FUNCTION_BLOCK Stage21 (* Template for a Basic Function Block Type *)
  (* Standard: 61499-2 *)
  (* Version 1.0, 2021-06-20, HP *)
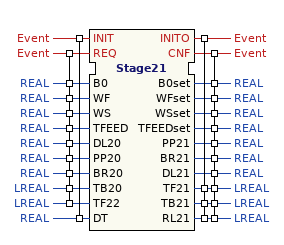
  EVENT_INPUT
    INIT WITH DT; (* Initialization Request *)
    REQ WITH WF, WS, TFEED, DL20, PP20, BR20, TB20, TF22, B0; (* Normal Execution Request *)
  END_EVENT
  EVENT_OUTPUT
    INITO WITH TB21, RL21, TF21; (* Initialization Confirm *)
    CNF WITH TB21, DL21, TF21, BR21, PP21, TFEEDset, WFset, WSset, RL21, B0set; (* Execution Confirmation *)
  END_EVENT
  VAR_INPUT
    B0 : REAL;
    WF : REAL;
    WS : REAL;
    TFEED : REAL;
    DL20 : REAL;
    PP20 : REAL;
    BR20 : REAL;
    TB20 : LREAL;
    TF22 : LREAL;
    DT : REAL;
  END_VAR
  VAR_OUTPUT
    B0set : REAL;
    WFset : REAL;
    WSset : REAL;
    TFEEDset : REAL;
    PP21 : REAL;
    BR21 : REAL;
    DL21 : REAL;
    TF21 : LREAL;
    TB21 : LREAL;
    RL21 : LREAL;
  END_VAR
  VAR
    AB : REAL; (* internal variabel *)
    UU : REAL;
    TREF : REAL;
    AD : REAL;
    AHC : REAL;
    AHR : REAL;
    AS : REAL;
    REC : REAL;
    WN : REAL;
    WN_1 : REAL;
    XKN : REAL;
    C1 : REAL;
    HS : REAL;
    G : REAL;
    W1 : REAL;
    TFREC : REAL;
    TS : REAL;
    DTS : REAL;
    TF21_last : REAL;
    RL21_last : REAL;
    TB21_last : REAL;
    USS : REAL;
    RHOB : REAL;
    CPB : REAL;
    CPF : REAL;
    FMW : REAL;
    HLV : REAL;
    HV : REAL;
    BPR : REAL;
    FMC : REAL;
    U : REAL;
    A : REAL;
    B : REAL;
    C : REAL;
    D1 : REAL;
    d : REAL;
    a : REAL;
    A1 : REAL;
    A2 : REAL;
    A3 : REAL;
    A4 : REAL;
    A5 : REAL;
    A6 : REAL;
    p : REAL;
    q : REAL;
    TC : REAL;
    PC : REAL;
    DTB21 : REAL;
    DEN21 : REAL;
    DH21 : REAL;
    DP21 : REAL;
    DPDH21 : REAL;
    DT21 : REAL;
    m : REAL;
    n : REAL;
    VR21 : REAL;
    DELTA21 : REAL;
    DELTA43 : REAL;
    DELTA65 : REAL;
    DELTA21_last : REAL;
    DELTA43_last : REAL;
    DELTA65_last : REAL;
  END_VAR
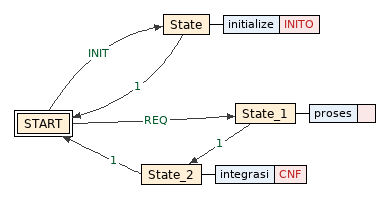
  EC_STATES
    START; (* Initial State *)
    State : initialize -> INITO;
    State_1 : proses;
    State_2 : integrasi -> CNF;
  END_STATES
  EC_TRANSITIONS
    START TO State := INIT;
    State TO START := 1;
    START TO State_1 := REQ;
    State_1 TO State_2 := 1;
    State_2 TO START := 1;
  END_TRANSITIONS
  ALGORITHM initialize IN ST: (* Initialization algorithm *)
TREF :=273.15;
AB :=57.2727;
AHC :=4069.2;
AHR :=2639.7;
AS :=3225.7;
REC :=0.0;
//TF2:=TF2;

//TFEED :=TFEED1+TREF;
 //TS:=TS1+TREF;
WN :=3.0;
XKN :=0.68;
HS:=0.11;
G :=9.81;
W1 :=0.50;

RL21 := 0.629413415201625;
TB21 := 316.382499320632;
TF21 := 312.855009206396;
TF22 := 310.669094657679;



RL21_last :=RL21;
TB21_last :=TB21;
TF21_last :=TF21;
  END_ALGORITHM
  ALGORITHM proses IN ST: (* kalkulasi *)
UU := TFEED;
U :=UU;

USS :=49.767;
C1 :=0.625;
RHOB :=1032.4; //maassa jenis brine
CPB :=1.00; //heatcapacity Brine
CPF :=1.00; //heat capacity feed
FMW :=23654.0;
HLV :=563.7959;
HV :=625.1971;
BPR :=2.192;
FMC :=34736.09;
//U :=UU; //feed temp



///  Calculate the physical properties

//A :=3.2437814;
//B :=5.86826*0.001;
//C :=1.1702379*0.00000001;
//D1 :=2.1878462*0.001;
//TC :=647.27;
//PC :=218.167;


A1 :=3.2437814;
A2:=5.86826*0.001;
A3:=1.1702379*0.00000001;
A4 :=2.1878462*0.001;
A5 :=647.27;
A6 :=218.167;

DTB21 :=A5-TB21;
DEN21 :=(A1+A2*DTB21+A3*DTB21*DTB21*DTB21)/(1+A4*DTB21)*DTB21/TB21;
p:=DEN21;
q:=10.0;
PP21 :=A6/(EXPT(q, p));

// calculate the brine flow rates
DP21:=PP20-PP21;
DH21:=RL21-C1*HS;
DPDH21 :=DP21*101000+G*RHOB*DH21;
m:=DPDH21*RHOB;
n:=0.5;
BR21 :=WN*XKN*RL21*(EXPT(m, n));
BR21 :=BR21*60.0/1000.0;

// calculate the vapor flow rates

DT21 :=TB21-BPR/1.8-(TF22+TF21)*0.5;
VR21:=U*AHR*DT21/HLV/1000.0;
DL21 :=DL20+VR21;


//// state equation
DELTA21 :=(BR20-BR21-VR21)*1000.0/RHOB/AB;
DELTA43 :=((BR20*CPB*(TB20-TB21))-VR21*(HV-CPB*(TB21-TREF)))*1000.0/AB/RHOB/CPB/RL21;
DELTA65 :=(WF*CPF*(TF22-TF21)*1000+(U*AHR*DT21))/FMW/CPF;
  END_ALGORITHM
  ALGORITHM integrasi IN ST: (* new algorithm *)
B0set:=B0;
WFset:=WF;
WSset:=WS ;
TFEEDset:=TFEED;
//integrasi
RL21 := (DELTA21 + DELTA21_last)*0.5*DT + RL21_last;
DELTA21_last :=DELTA21 ;
RL21_last :=RL21;

TB21:= (DELTA43 + DELTA43_last)*0.5*DT + TB21_last;
DELTA43_last :=DELTA43 ;
TB21_last:=TB21;

TF21 := (DELTA65 + DELTA65_last)*0.5*DT + TF21_last;
DELTA65_last :=DELTA65 ;
TF21_last :=TF21;
  END_ALGORITHM
END_FUNCTION_BLOCK
